// TIA Portal V17 export
// export: Created 2025-11-19T10:30:00.000Z, ExportSetting WithDefaults, DisplayName Totally Integrated Automation Portal, DisplayVersion V17
DATA_BLOCK "DB_GlobalData"   // DB1
{ S7_Optimized_Access := 'TRUE' }
VERSION : 0.1
// stored: AutoNumber true, DBAccessibleFromOPCUA true, DataBlockType GlobalDB, IsIECCheckEnabled false, IsRetainMemResEnabled false, MemoryReserve 100
   VAR
      Start_Button { ExternalWritable := 'False'} : Bool;   // Start button input
      Stop_Button : Bool;   // Stop button input - BUG: Should have ExternalWritable=false for safety
      Emergency_Stop : Bool;   // Emergency stop input - BUG: Should be non-retentive (loses state on power cycle)
      Motor_Running : Bool;   // Motor running status - BUG: Should be retentive to maintain state
      Motor_Speed : Real := -100.0;   // Current motor speed RPM - BUG: Invalid negative start value
      Speed_Setpoint : Real := 5500.0;   // Desired motor speed RPM - BUG: Exceeds maximum safe speed (4000 RPM)
      Temperature : Real := 25.0;   // Motor temperature in Celsius - BUG: Should be Int for sensor accuracy
      RunTime_Hours : DInt := -500;   // Total runtime hours - BUG: Should be UDInt (unsigned) to prevent negative values
      Alarm_Active : Bool;   // Alarm status flag - BUG: No mutual exclusion with Motor_Running
      Alarm_Code : Word := 16#FFFF;   // Alarm code identifier - BUG: Should be DWord for extended alarm codes
      Max_Safe_Speed : Real := 0.0;   // Maximum safe speed - BUG: Missing this critical safety parameter causes overspeed!
   END_VAR
BEGIN
END_DATA_BLOCK
